// TwinCAT 3 PLC project HMIVisuPopum
// ProgramVersion: 3.1.4024.0
// libraries:
//   CmpBitmapPool, * (System)
//   Tc2_Standard, * (Beckhoff Automation GmbH)
//   Tc2_System, * (Beckhoff Automation GmbH)
//   Tc3_Module, * (Beckhoff Automation GmbH)
//   VisuSymbols,3.5.10.0,System
// project tree:
//   / GlobalTextList.TcGTLO, PlcTask.TcTTO, Visualization Manager.TcVMO (not stored), VISU_TASK.TcTTO
//   GVLs/ GVL.TcGVL
//   POUs/ MAIN.TcPOU, OpenMessageDialogEmergency.TcPOU, popup.TcPOU
//   VISUs/ image.TcIPO (not stored), Main.TcVIS, Popup.TcVIS
// real-time tasks:
//   TASK PlcTask: cycle T#10ms, priority 20, ADS port 350
//   TASK VISU_TASK: cycle T#200000us, priority 30, ADS port 351

CONFIGURATION HMIVisuPopum
    RESOURCE PLC ON TwinCAT3
        TASK PlcTask(INTERVAL := T#10ms, PRIORITY := 20);
        TASK VISU_TASK(INTERVAL := T#200000us, PRIORITY := 30);
        PROGRAM MAIN WITH PlcTask : MAIN;
        PROGRAM VisuElems_Visu_Prg WITH VISU_TASK : VisuElems.Visu_Prg;
    END_RESOURCE
END_CONFIGURATION

// ---- GVLs/GVL.TcGVL
{attribute 'qualified_only'}
VAR_GLOBAL
	emergency: BOOL;
	iDialogManager : VisuElems.IDialogManager;
	iMessageDialog : VisuElems.IVisualisationDialog;
END_VAR

// ---- POUs/MAIN.TcPOU
PROGRAM MAIN
VAR
END_VAR

popup();

END_PROGRAM

// ---- POUs/popup.TcPOU
PROGRAM popup
VAR
	fbOpenMessageDialogEmergency: R_trig;
END_VAR

fbOpenMessageDialogEmergency(CLK := gvl.emergency);
IF fbOpenMessageDialogEmergency.Q  THEN
	OpenMessageDialogEmergency();
END_IF

END_PROGRAM

// ---- POUs/OpenMessageDialogEmergency.TcPOU
FUNCTION OpenMessageDialogEmergency : BOOL
VAR_INPUT
END_VAR
VAR
	stMyRect : VisuElems.VisuStructSimpleRectangle;
	pTempClientData : POINTER TO VisuElems.VisuStructClientData;
	pLastClientData : POINTER TO VisuElems.VisuStructClientData;
	nIteratorSave : INT;
	nCounter : INT;
END_VAR

nIteratorSave := VisuElems.VisuElemBase.Visu_Globals.g_ClientManager.SaveIteration(); 
VisuElems.VisuElemBase.Visu_Globals.g_ClientManager.BeginIteration();

GVL.iDialogManager := VisuElems.VisuElemBase.g_VisuManager.GetDialogManager();

// Assign the argument in all currently active clients
pTempClientData := VisuElems.VisuElemBase.Visu_Globals.g_ClientManager.GetNextClient();

// Open Dialog on all Clients
GVL.iMessageDialog := GVL.iDialogManager.GetDialog('Popup'); // dialog to be handled is specified
IF GVL.iMessageDialog <> 0 THEN
	stMyRect.ptTopLeft.iX := 200;
	stMyRect.ptTopLeft.iY := 100;
	stMyRect.ptBottomRight.iX := 200;
	stMyRect.ptBottomRight.iY := 450;
	GVL.iDialogManager.OpenDialog3(GVL.iMessageDialog, pTempClientData, TRUE, ADR(stMyRect), 0, VisuElems.Visu_InputFlags.GlobalOpenCloseDialog);
END_IF

VisuElems.VisuElemBase.Visu_Globals.g_ClientManager.RestoreIteration(nIteratorSave);

END_FUNCTION

// ---- GlobalTextList.TcGTLO
TEXTLIST GlobalTextList
  377 = 'Close'
  193 = 'Emergency Button'
END_TEXTLIST

// ---- VISUs/Main.TcVIS
VISUALIZATION Main  // 800x480
END_VISUALIZATION

// ---- VISUs/Popup.TcVIS
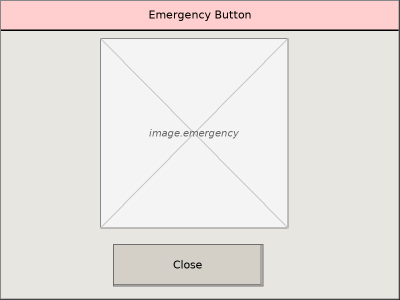
VISUALIZATION Popup  // 400x300
    Rectangle (0,0 400x30), "Emergency Button"
    Rectangle (0,30 400x270)
    Image (100,38 188x190), image: image.emergency
    Button (113,244 150x42), "Close"
        OnMouseClick: CloseDialog Dialog=Popup, Result=OK, NumpadKeypadSet=True
END_VISUALIZATION
